// TIA Portal V18 export
DATA_BLOCK "DB_Recipe"   // DB290
{ S7_Optimized_Access := 'TRUE' }
VERSION : 0.1
// stored: AutoNumber true, DBAccessibleFromOPCUA true, IsOnlyStoredInLoadMemory false, IsRetainMemResEnabled false, IsWriteProtectedInAS false, MemoryReserve 100
   VAR
      HMI_Recipe : Int := 0;
      HMI_Recipe_Data : String := '';
      Recepie_name : String;
   END_VAR
BEGIN
END_DATA_BLOCK
